TYPE ST_KKKW_Zustand :
STRUCT

	Betrieb_Anford		: BOOL;
	Betrieb_Soll		: BOOL;
	Betrieb				: BOOL;

	Freigabe			: BOOL;
	Freigabe_Deakt		: BOOL;
	Freigabe_Code		: WORD;
	Stoerung			: BOOL;

	Anforderung_Pumpe_Netz	: BOOL;
	CompressorSpeed : DINT;

	Stoerung_Code		: WORD;

	Warnung				: BOOL;
	Warnung_Code		: WORD;
END_STRUCT
END_TYPE

(* stored: Version 1.1.0.1, ProductVersion 3.1.4024.9
   DUT ST_KKKW_Zustand: Id {9954594e-090d-4690-8a2c-0456da581ab1} *)
